// TIA Portal V17 export
// export: Created 2023-12-22T15:04:42.9344421Z, ExportSetting WithDefaults, DisplayName Totally Integrated Automation Portal, DisplayVersion V17, DisplayName TIA Portal Openness, DisplayVersion V17, DisplayName TIA Portal Version Control Interface, DisplayVersion V17, DisplayName STEP 7 Professional, DisplayVersion V17, DisplayName STEP 7 Safety, DisplayVersion V17, DisplayName WinCC Advanced, DisplayVersion V17
FUNCTION "drv_INV" : Void   // FC111, LAD
{ S7_Optimized_Access := 'FALSE' }
VERSION : 0.1
// stored: AutoNumber false, IsIECCheckEnabled false, SetENOAutomatically false, UDAEnableTagReadback false
   VAR_INPUT
      S : Bool;   // Сигнал
      I : Bool;   // Инверсия
   END_VAR
   VAR_IN_OUT
      R : Bool;   // Результат
   END_VAR
BEGIN

REGION Network 1: Инверсия сигнала
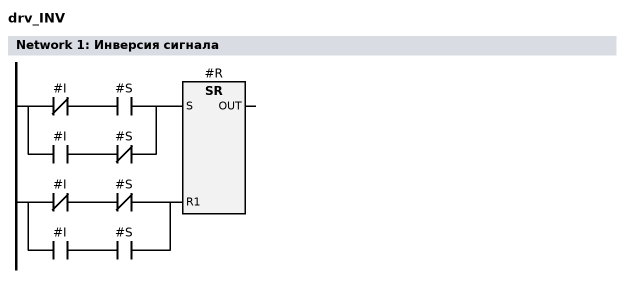
   RUNG wire#powerrail
      I_Contact( #I )
      Contact( #S )
      wire#w1
      S_SR(operand := #R, r1 := wire#w2)
   END_RUNG
   RUNG wire#powerrail
      Contact( #I )
      I_Contact( #S )
   END_RUNG wire#w1
   RUNG wire#powerrail
      I_Contact( #I )
      I_Contact( #S )
   END_RUNG wire#w2
   RUNG wire#powerrail
      Contact( #I )
      Contact( #S )
   END_RUNG wire#w2
   // the same network as SCL:
   IF (NOT #I AND #S) OR (#I AND NOT #S) THEN
       #R := TRUE;   // SR flip-flop
   END_IF;
   IF (NOT #I AND NOT #S) OR (#I AND #S) THEN #R := FALSE; END_IF;
END_REGION
END_FUNCTION
